FUNCTION_BLOCK RQST_GEN (* FBMGT Request Generator *)
  (* Standard: 61499 ITA; ApplicationDomain: Device Management; Function: FBMGT Request Generator *)
  (* Version 0.0, 2001-11-27, JHC, Rockwell Automation, Copied/modified from QUERY_GEN. *)
  (* Compiler header: package fb.rt.ita; *)
  (* Compiler Java IBM VisualAge 3.0 *)
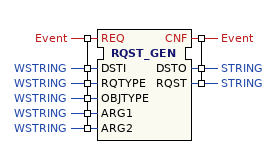
  EVENT_INPUT
    REQ WITH DSTI, RQTYPE, OBJTYPE, ARG1, ARG2;
  END_EVENT
  EVENT_OUTPUT
    CNF WITH DSTO, RQST;
  END_EVENT
  VAR_INPUT
    DSTI : WSTRING; (* Destination *)
    RQTYPE : WSTRING; (* CREATE,DELETE,READ,WRITE,QUERY *)
    OBJTYPE : WSTRING; (* FB,Connection *)
    ARG1 : WSTRING; (* FB Name or Connection Source *)
    ARG2 : WSTRING; (* FB Type or Connection Destination *)
  END_VAR
  VAR_OUTPUT
    DSTO : STRING; (* DSTI converted to STRING *)
    RQST : STRING; (* FBMGT request *)
  END_VAR
END_FUNCTION_BLOCK
